FUNCTION FunLadoTrabajoCaballete : Uint
VAR_INPUT
	Piezas_LadoA 			: UINT ;
	Piezas_Ladob			: UINT ;
	Recoger					: BOOL;
	Dejar					: BOOL ;
	GestionLadoTrabajo		: INT ;
	
END_VAR
VAR
	DifPiezas 				: UINT;
	
END_VAR

IF  Dejar AND GestionLadoTrabajo = 0 THEN 
  
	IF Piezas_LadoA = 0 AND Piezas_Ladob =0 THEN 
		FunLadoTrabajoCaballete := 0 ;
	
	ELSIF Piezas_LadoA <> Piezas_Ladob THEN 
		DifPiezas := ABS (Piezas_LadoA - Piezas_Ladob) ;
			IF DifPiezas > 1 AND Piezas_LadoA > Piezas_Ladob THEN 
				FunLadoTrabajoCaballete := 180 ;
			ELSIF DifPiezas > 1 AND Piezas_Ladob > Piezas_LadoA	THEN
				FunLadoTrabajoCaballete := 0 ;
			END_IF
	END_IF
		
	IF DifPiezas = 1   THEN
			IF  Piezas_Ladob < Piezas_LadoA THEN 
				FunLadoTrabajoCaballete := 180 ;
			ELSIF Piezas_LadoA < Piezas_LadoB THEN 
				FunLadoTrabajoCaballete := 0 ;
			END_IF
	END_IF
END_IF

IF  Recoger AND GestionLadoTrabajo = 0 THEN 
  
	IF Piezas_LadoA = Piezas_Ladob  THEN 
		FunLadoTrabajoCaballete := 180 ;
	
	ELSIF Piezas_LadoA <> Piezas_Ladob THEN 
		DifPiezas := ABS (Piezas_LadoA - Piezas_Ladob) ;
			IF DifPiezas > 1 AND Piezas_LadoA > Piezas_Ladob THEN 
				FunLadoTrabajoCaballete := 0 ;
			ELSIF DifPiezas > 1 AND Piezas_Ladob > Piezas_LadoA	THEN
				FunLadoTrabajoCaballete := 180 ;
			END_IF
	END_IF
		
	IF DifPiezas = 1   THEN
			IF  Piezas_Ladob < Piezas_LadoA THEN 
				FunLadoTrabajoCaballete := 00 ;
			ELSIF Piezas_LadoA < Piezas_LadoB THEN 
				FunLadoTrabajoCaballete := 180 ;
			END_IF
	END_IF
END_IF

IF GestionLadoTrabajo <> 0 THEN
	IF GestionLadoTrabajo = 1 THEN
		FunLadoTrabajoCaballete := 0 ;
	ELSIF GestionLadoTrabajo = 2 THEN 
		FunLadoTrabajoCaballete := 180 ;	
	END_IF
	


END_IF

END_FUNCTION

(* stored: Version 1.1.0.1, ProductVersion 3.1.4024.11
   POU FunLadoTrabajoCaballete: Id {03154322-5f1d-40a2-be63-9f98acb46263}, SpecialFunc None *)
